(* CODESYS project EVL.gvl.xml

Project tree, tasks and I/O mapping:
  global variables EVL
*)

// EVL
(* THIS EVL IS AUTOGENERATED. DO NOT MODIFY THESE ATTRIBUTES. *)
{attribute 'location' := '16#800' }
{attribute 'linkalways'}
{attribute 'qualified_only'}
VAR_GLOBAL

END_VAR
